// TIA Portal V15.1 export
// export: Created 2024-06-21T08:41:25.7008417Z, ExportSetting WithDefaults, DisplayName Totally Integrated Automation Portal, DisplayVersion V15.1 Update 5, DisplayName TIA Portal Openness, DisplayVersion V15.1 Update 5, DisplayName SINAMICS Startdrive Advanced, DisplayVersion V15.1, DisplayName G130, G150, S120, S150, SINAMICS MV, S210, DisplayVersion V15.1, DisplayName G110M, G120, G120C, G120D, G120P, DisplayVersion V15.1, DisplayName STEP 7 Professional, DisplayVersion V15.1 Update 5, DisplayName STEP 7 Safety, DisplayVersion V15.1, DisplayName WinCC Professional, DisplayVersion V15.1 Update 5, DisplayName SIMATIC Visualization Architect, DisplayVersion V15.1
FUNCTION "DPComPLC212" : Void   // FC261, FBD
TITLE = DPComPLC212
{ S7_Optimized_Access := 'FALSE' }
AUTHOR : VCG
FAMILY : LocFncGn
NAME : 211Intf
VERSION : 0.1
// stored: AutoNumber false, IsIECCheckEnabled false, SetENOAutomatically False, UDAEnableTagReadback false
   VAR_OUTPUT
      O_AlarmA : Bool;   // Alarm A
      O_AlarmB : Bool;   // Alarm B
      O_AlarmC : Bool;   // Alarm C
      O_AlarmD : Bool;   // Alarm D
      O_AlarmABCondition : Bool;   // Alarms resetable
      H_IAnim : Word;   // For animation of icon
   END_VAR
   VAR_TEMP
      TempInt : Int;
   END_VAR
BEGIN

REGION Network 1: **** --------------------- R228.01 --> 210CR23 --------------------- ****
END_REGION

REGION Network 2: **** 1 - Inputs **** 212A - Access Stop Request
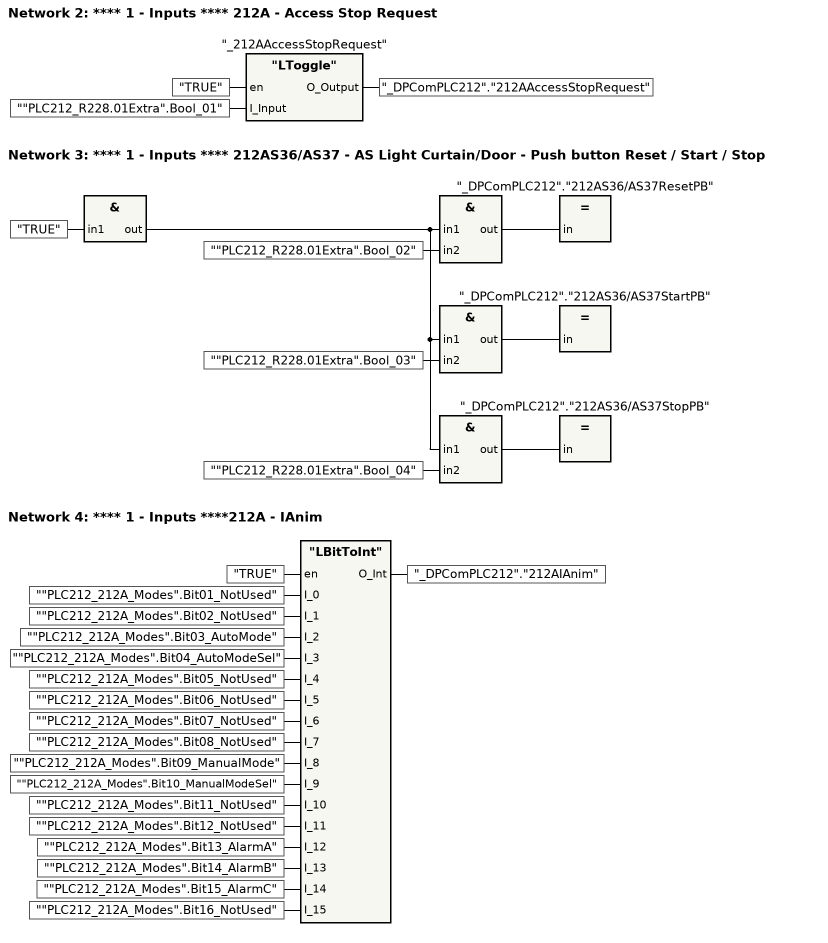
   // no checked SCL form for this network; see the picture
END_REGION

REGION Network 3: **** 1 - Inputs **** 212AS36/AS37 - AS Light Curtain/Door - Push button Reset / Start / Stop
   // no checked SCL form for this network; see the picture
END_REGION

REGION Network 4: **** 1 - Inputs ****212A - IAnim
   // no checked SCL form for this network; see the picture
END_REGION

REGION Network 5: **** 1 - Inputs **** 212A - Modes
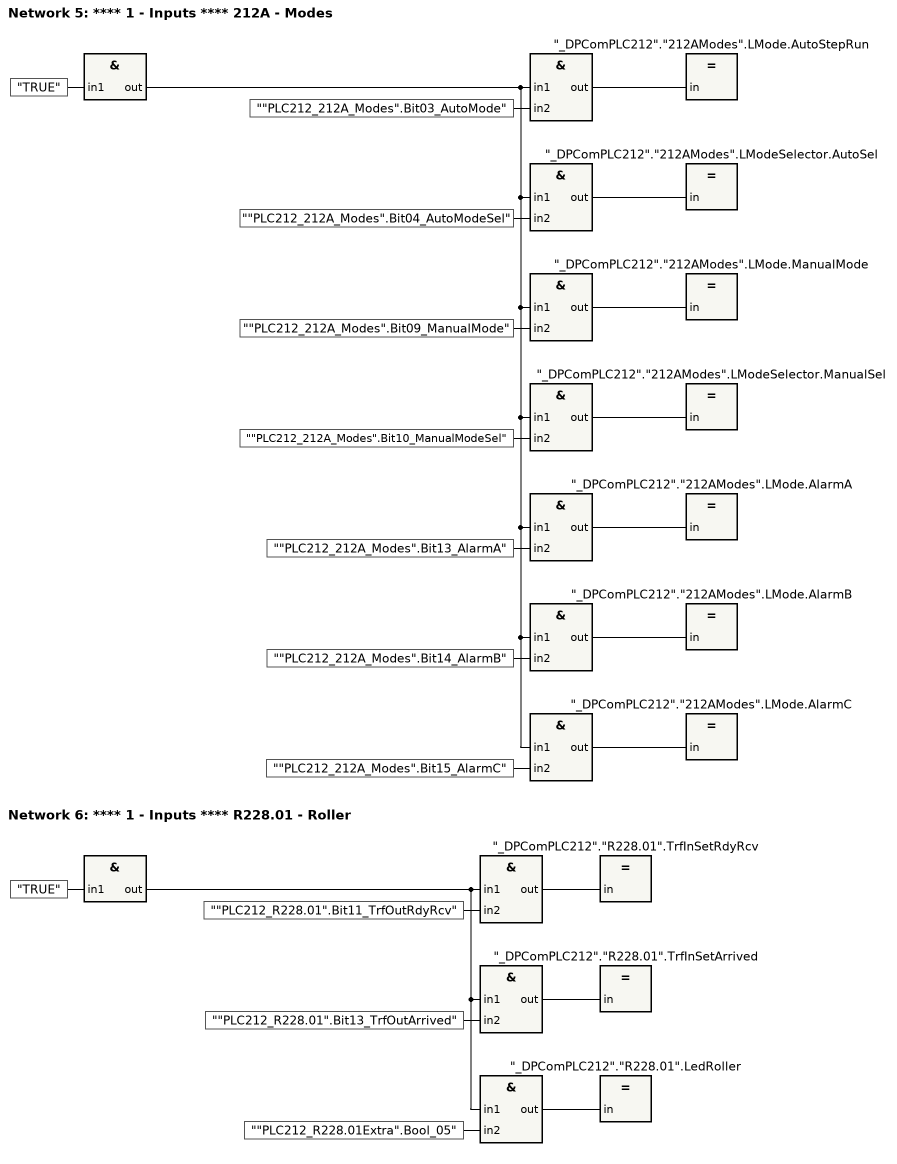
   // no checked SCL form for this network; see the picture
END_REGION

REGION Network 6: **** 1 - Inputs **** R228.01 - Roller
   // no checked SCL form for this network; see the picture
END_REGION

REGION Network 7: **** --------------------- R228.02 --> 220CR23 --------------------- ****
END_REGION

REGION Network 8: **** 1 - Inputs **** 212AS38/AS39 - AS Light Curtain/Door - Push button Reset / Start / Stop
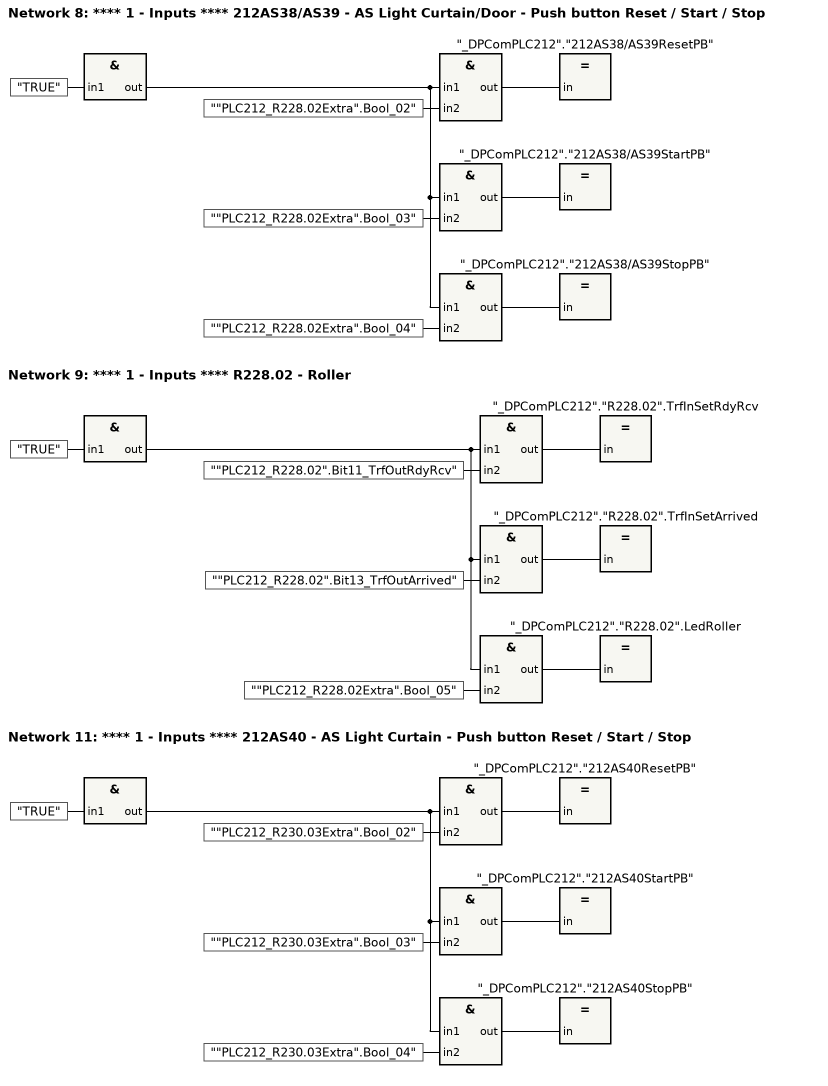
   // no checked SCL form for this network; see the picture
END_REGION

REGION Network 9: **** 1 - Inputs **** R228.02 - Roller
   // no checked SCL form for this network; see the picture
END_REGION

REGION Network 10: **** --------------------- R230.03 --> 230CA21 --------------------- ****
END_REGION

REGION Network 11: **** 1 - Inputs **** 212AS40 - AS Light Curtain - Push button Reset / Start / Stop
   // no checked SCL form for this network; see the picture
END_REGION

REGION Network 12: **** 1 - Inputs ****212D - IAnim
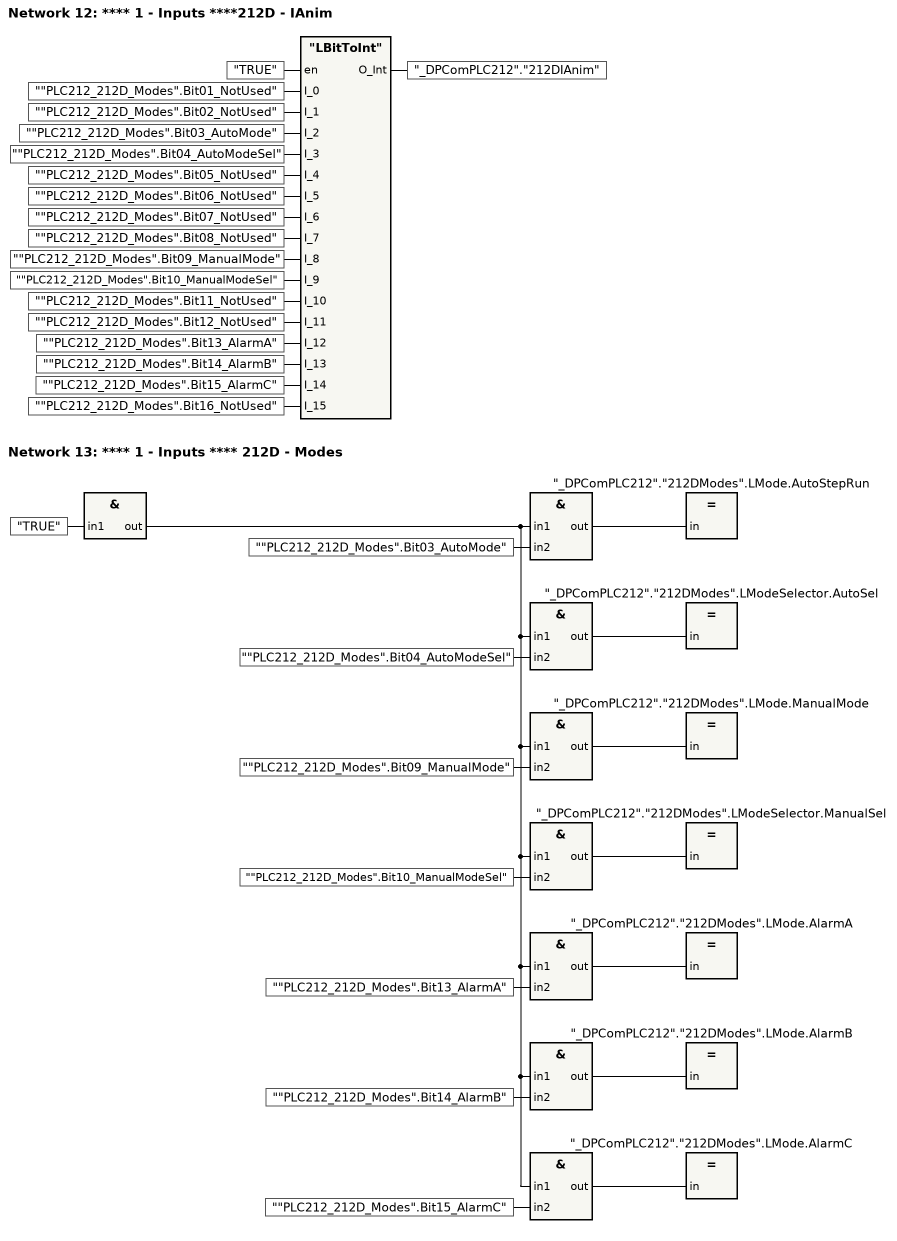
   // no checked SCL form for this network; see the picture
END_REGION

REGION Network 13: **** 1 - Inputs **** 212D - Modes
   // no checked SCL form for this network; see the picture
END_REGION

REGION Network 14: **** 1 - Inputs **** R230.03 - Roller
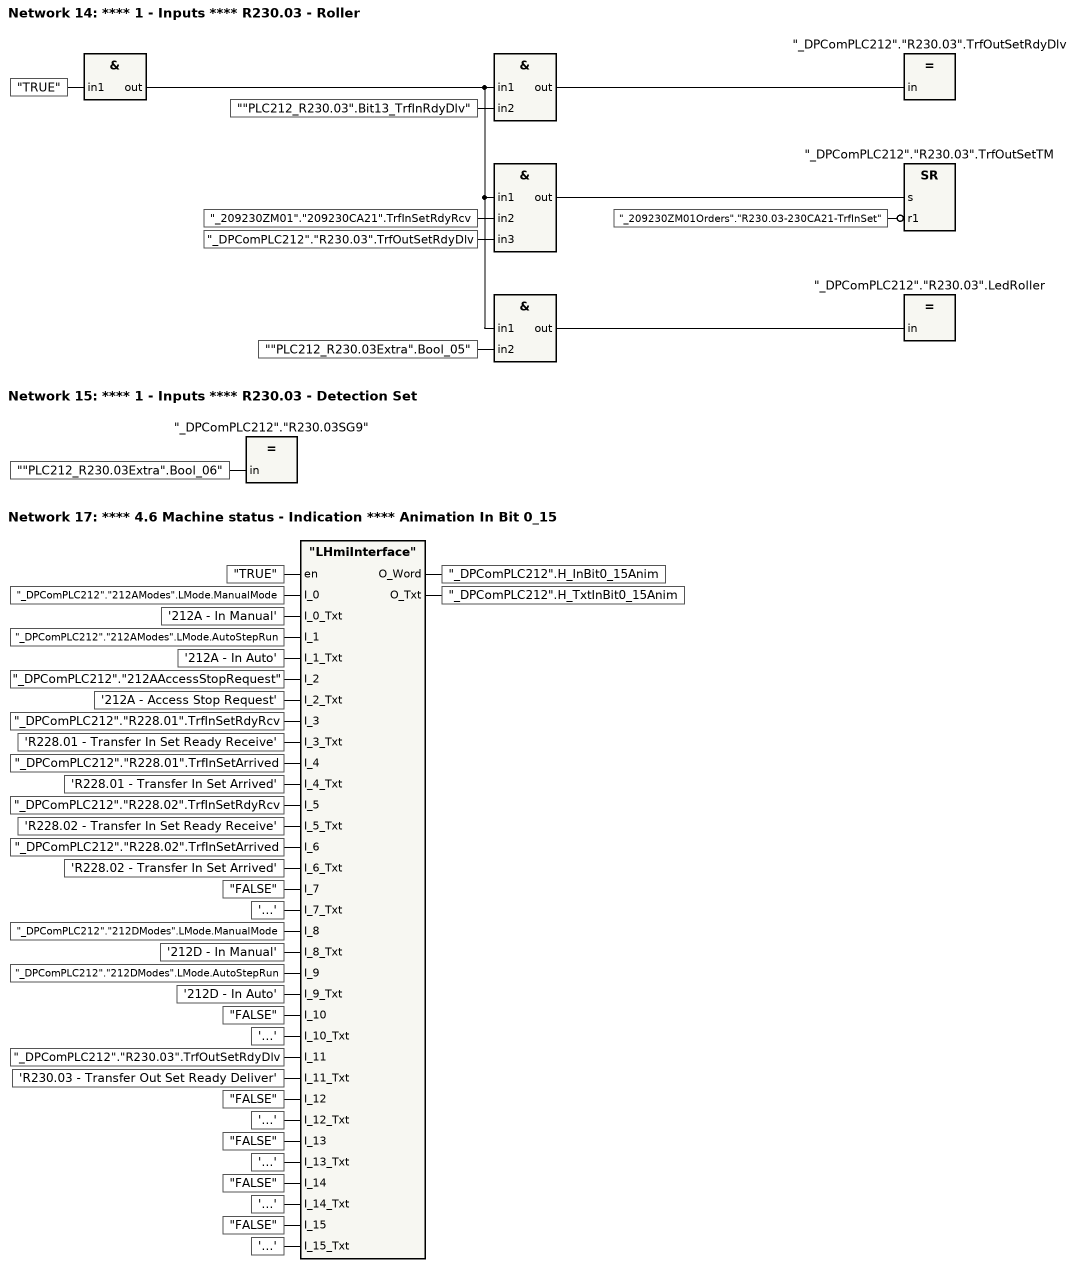
   // no checked SCL form for this network; see the picture
END_REGION

REGION Network 15: **** 1 - Inputs **** R230.03 - Detection Set
   // no checked SCL form for this network; see the picture
END_REGION

REGION Network 16: **** -------------------------------------------------- ****
END_REGION

REGION Network 17: **** 4.6 Machine status - Indication **** Animation In Bit 0_15
   // H_In0_15Anim
   IF "TRUE" THEN
       "LHmiInterface"(I_0 := "_DPComPLC212"."212AModes".LMode.ManualMode,
                       I_0_Txt := '212A - In Manual',
                       I_1 := "_DPComPLC212"."212AModes".LMode.AutoStepRun,
                       I_1_Txt := '212A - In Auto',
                       I_2 := "_DPComPLC212"."212AAccessStopRequest",
                       I_2_Txt := '212A - Access Stop Request',
                       I_3 := "_DPComPLC212"."R228.01".TrfInSetRdyRcv,
                       I_3_Txt := 'R228.01 - Transfer In Set Ready Receive',
                       I_4 := "_DPComPLC212"."R228.01".TrfInSetArrived,
                       I_4_Txt := 'R228.01 - Transfer In Set Arrived',
                       I_5 := "_DPComPLC212"."R228.02".TrfInSetRdyRcv,
                       I_5_Txt := 'R228.02 - Transfer In Set Ready Receive',
                       I_6 := "_DPComPLC212"."R228.02".TrfInSetArrived,
                       I_6_Txt := 'R228.02 - Transfer In Set Arrived',
                       I_7 := "FALSE",
                       I_7_Txt := '...',
                       I_8 := "_DPComPLC212"."212DModes".LMode.ManualMode,
                       I_8_Txt := '212D - In Manual',
                       I_9 := "_DPComPLC212"."212DModes".LMode.AutoStepRun,
                       I_9_Txt := '212D - In Auto',
                       I_10 := "FALSE",
                       I_10_Txt := '...',
                       I_11 := "_DPComPLC212"."R230.03".TrfOutSetRdyDlv,
                       I_11_Txt := 'R230.03 - Transfer Out Set Ready Deliver',
                       I_12 := "FALSE",
                       I_12_Txt := '...',
                       I_13 := "FALSE",
                       I_13_Txt := '...',
                       I_14 := "FALSE",
                       I_14_Txt := '...',
                       I_15 := "FALSE",
                       I_15_Txt := '...',
                       O_Word => "_DPComPLC212".H_InBit0_15Anim,
                       O_Txt => "_DPComPLC212".H_TxtInBit0_15Anim);
   END_IF;
END_REGION

REGION Network 18: **** 4.6 Machine status - Indication **** Animation In Bit 16_31
   // H_In16_31Anim
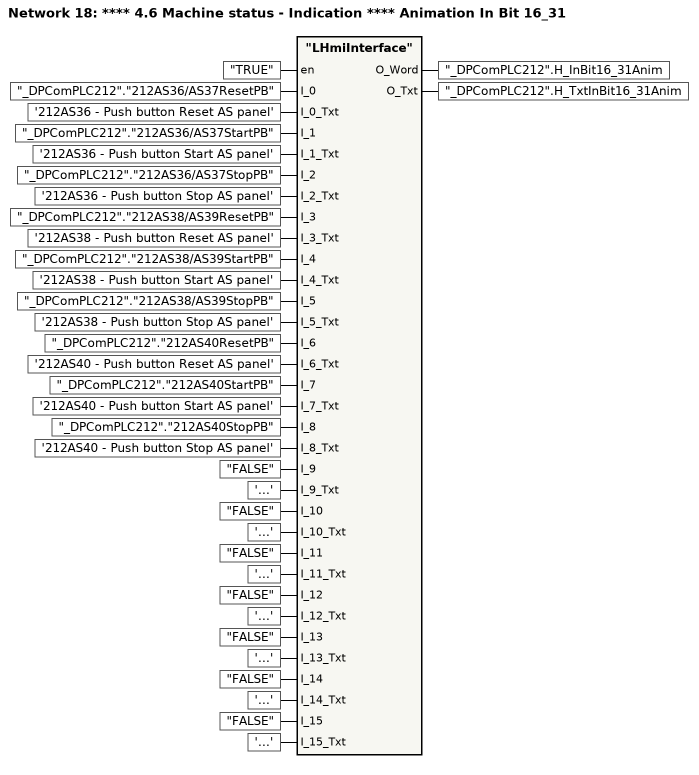
   IF "TRUE" THEN
       "LHmiInterface"(I_0 := "_DPComPLC212"."212AS36/AS37ResetPB",
                       I_0_Txt := '212AS36 - Push button Reset AS panel',
                       I_1 := "_DPComPLC212"."212AS36/AS37StartPB",
                       I_1_Txt := '212AS36 - Push button Start AS panel',
                       I_2 := "_DPComPLC212"."212AS36/AS37StopPB",
                       I_2_Txt := '212AS36 - Push button Stop AS panel',
                       I_3 := "_DPComPLC212"."212AS38/AS39ResetPB",
                       I_3_Txt := '212AS38 - Push button Reset AS panel',
                       I_4 := "_DPComPLC212"."212AS38/AS39StartPB",
                       I_4_Txt := '212AS38 - Push button Start AS panel',
                       I_5 := "_DPComPLC212"."212AS38/AS39StopPB",
                       I_5_Txt := '212AS38 - Push button Stop AS panel',
                       I_6 := "_DPComPLC212"."212AS40ResetPB",
                       I_6_Txt := '212AS40 - Push button Reset AS panel',
                       I_7 := "_DPComPLC212"."212AS40StartPB",
                       I_7_Txt := '212AS40 - Push button Start AS panel',
                       I_8 := "_DPComPLC212"."212AS40StopPB",
                       I_8_Txt := '212AS40 - Push button Stop AS panel',
                       I_9 := "FALSE",
                       I_9_Txt := '...',
                       I_10 := "FALSE",
                       I_10_Txt := '...',
                       I_11 := "FALSE",
                       I_11_Txt := '...',
                       I_12 := "FALSE",
                       I_12_Txt := '...',
                       I_13 := "FALSE",
                       I_13_Txt := '...',
                       I_14 := "FALSE",
                       I_14_Txt := '...',
                       I_15 := "FALSE",
                       I_15_Txt := '...',
                       O_Word => "_DPComPLC212".H_InBit16_31Anim,
                       O_Txt => "_DPComPLC212".H_TxtInBit16_31Anim);
   END_IF;
END_REGION

REGION Network 19: **** 4.6 Machine status - Indication **** Animation Out Bit 0_15
   // H_Out0_15Anim
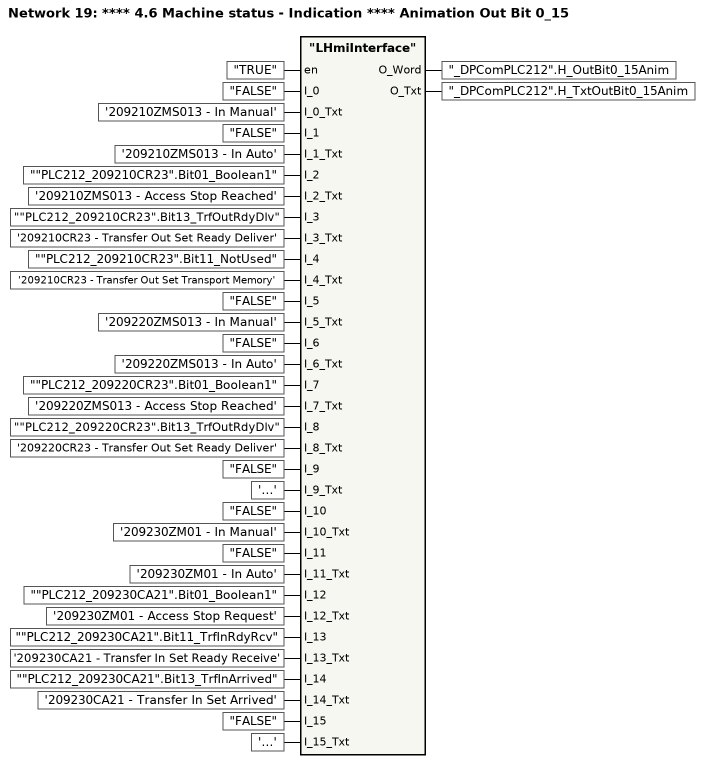
   // no checked SCL form for this network; see the picture
END_REGION

REGION Network 20: **** 4.6 Machine status - Indication **** Animation Out Bit 16_31
   // H_Out16_31Anim
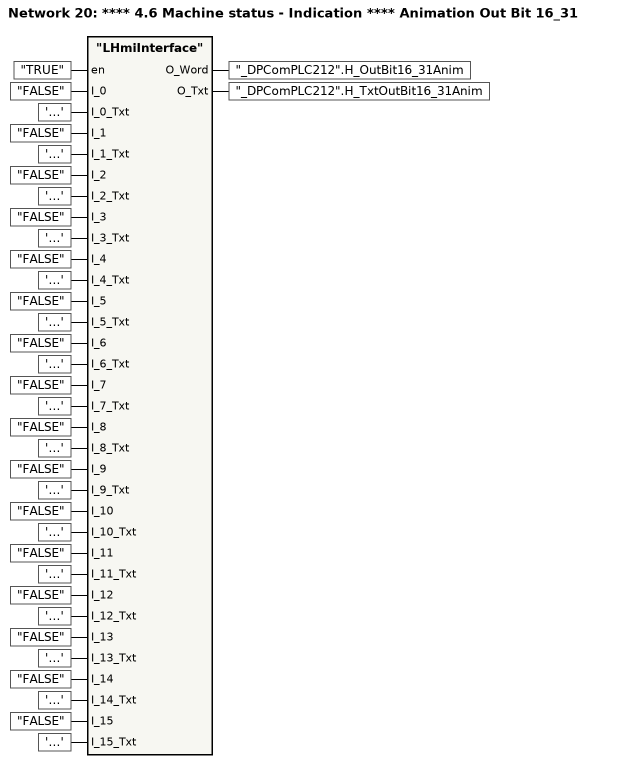
   IF "TRUE" THEN
       "LHmiInterface"(I_0 := "FALSE",
                       I_0_Txt := '...',
                       I_1 := "FALSE",
                       I_1_Txt := '...',
                       I_2 := "FALSE",
                       I_2_Txt := '...',
                       I_3 := "FALSE",
                       I_3_Txt := '...',
                       I_4 := "FALSE",
                       I_4_Txt := '...',
                       I_5 := "FALSE",
                       I_5_Txt := '...',
                       I_6 := "FALSE",
                       I_6_Txt := '...',
                       I_7 := "FALSE",
                       I_7_Txt := '...',
                       I_8 := "FALSE",
                       I_8_Txt := '...',
                       I_9 := "FALSE",
                       I_9_Txt := '...',
                       I_10 := "FALSE",
                       I_10_Txt := '...',
                       I_11 := "FALSE",
                       I_11_Txt := '...',
                       I_12 := "FALSE",
                       I_12_Txt := '...',
                       I_13 := "FALSE",
                       I_13_Txt := '...',
                       I_14 := "FALSE",
                       I_14_Txt := '...',
                       I_15 := "FALSE",
                       I_15_Txt := '...',
                       O_Word => "_DPComPLC212".H_OutBit16_31Anim,
                       O_Txt => "_DPComPLC212".H_TxtOutBit16_31Anim);
   END_IF;
END_REGION

REGION Network 21: **** 4.6 Machine status - Indication **** Animation Safety In Bit 0_15
   // H_FIn0_15Anim
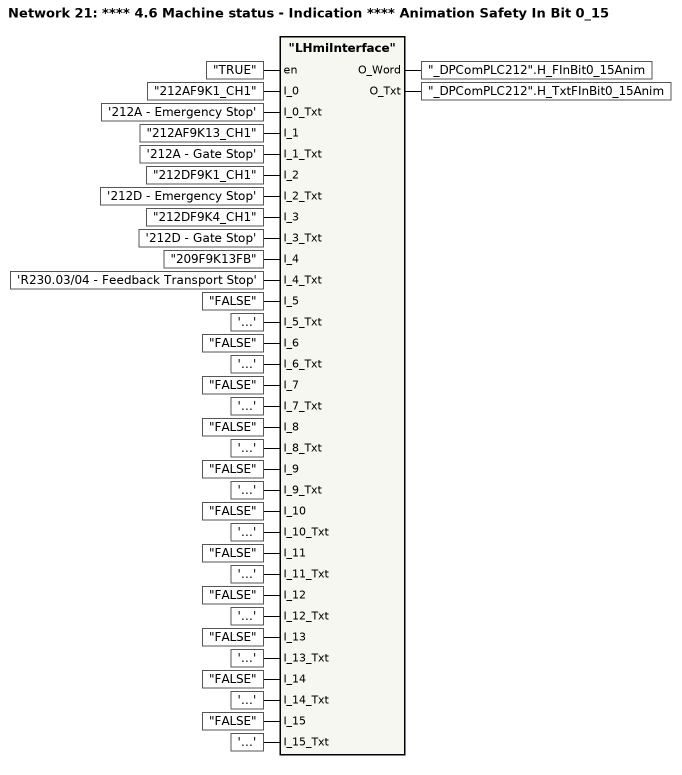
   IF "TRUE" THEN
       "LHmiInterface"(I_0 := "212AF9K1_CH1",
                       I_0_Txt := '212A - Emergency Stop',
                       I_1 := "212AF9K13_CH1",
                       I_1_Txt := '212A - Gate Stop',
                       I_2 := "212DF9K1_CH1",
                       I_2_Txt := '212D - Emergency Stop',
                       I_3 := "212DF9K4_CH1",
                       I_3_Txt := '212D - Gate Stop',
                       I_4 := "209F9K13FB",
                       I_4_Txt := 'R230.03/04 - Feedback Transport Stop',
                       I_5 := "FALSE",
                       I_5_Txt := '...',
                       I_6 := "FALSE",
                       I_6_Txt := '...',
                       I_7 := "FALSE",
                       I_7_Txt := '...',
                       I_8 := "FALSE",
                       I_8_Txt := '...',
                       I_9 := "FALSE",
                       I_9_Txt := '...',
                       I_10 := "FALSE",
                       I_10_Txt := '...',
                       I_11 := "FALSE",
                       I_11_Txt := '...',
                       I_12 := "FALSE",
                       I_12_Txt := '...',
                       I_13 := "FALSE",
                       I_13_Txt := '...',
                       I_14 := "FALSE",
                       I_14_Txt := '...',
                       I_15 := "FALSE",
                       I_15_Txt := '...',
                       O_Word => "_DPComPLC212".H_FInBit0_15Anim,
                       O_Txt => "_DPComPLC212".H_TxtFInBit0_15Anim);
   END_IF;
END_REGION

REGION Network 22: **** 4.6 Machine status - Indication **** Animation Safety Out Bit 0_15
   // H_FOut0_15Anim
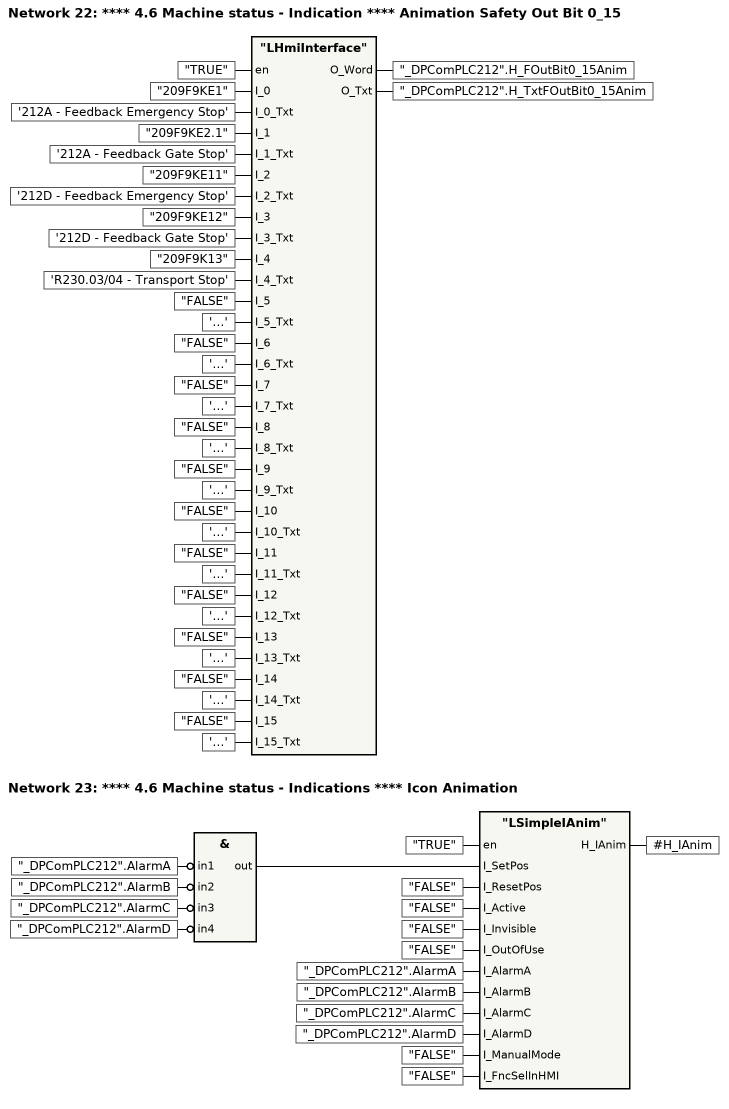
   IF "TRUE" THEN
       "LHmiInterface"(I_0 := "209F9KE1",
                       I_0_Txt := '212A - Feedback Emergency Stop',
                       I_1 := "209F9KE2.1",
                       I_1_Txt := '212A - Feedback Gate Stop',
                       I_2 := "209F9KE11",
                       I_2_Txt := '212D - Feedback Emergency Stop',
                       I_3 := "209F9KE12",
                       I_3_Txt := '212D - Feedback Gate Stop',
                       I_4 := "209F9K13",
                       I_4_Txt := 'R230.03/04 - Transport Stop',
                       I_5 := "FALSE",
                       I_5_Txt := '...',
                       I_6 := "FALSE",
                       I_6_Txt := '...',
                       I_7 := "FALSE",
                       I_7_Txt := '...',
                       I_8 := "FALSE",
                       I_8_Txt := '...',
                       I_9 := "FALSE",
                       I_9_Txt := '...',
                       I_10 := "FALSE",
                       I_10_Txt := '...',
                       I_11 := "FALSE",
                       I_11_Txt := '...',
                       I_12 := "FALSE",
                       I_12_Txt := '...',
                       I_13 := "FALSE",
                       I_13_Txt := '...',
                       I_14 := "FALSE",
                       I_14_Txt := '...',
                       I_15 := "FALSE",
                       I_15_Txt := '...',
                       O_Word => "_DPComPLC212".H_FOutBit0_15Anim,
                       O_Txt => "_DPComPLC212".H_TxtFOutBit0_15Anim);
   END_IF;
END_REGION

REGION Network 23: **** 4.6 Machine status - Indications **** Icon Animation
   // Animation for icon
   IF "TRUE" THEN
       "LSimpleIAnim"(I_SetPos := NOT "_DPComPLC212".AlarmA AND NOT "_DPComPLC212".AlarmB AND NOT "_DPComPLC212".AlarmC AND NOT "_DPComPLC212".AlarmD,
                      I_ResetPos := "FALSE",
                      I_Active := "FALSE",
                      I_Invisible := "FALSE",
                      I_OutOfUse := "FALSE",
                      I_AlarmA := "_DPComPLC212".AlarmA,
                      I_AlarmB := "_DPComPLC212".AlarmB,
                      I_AlarmC := "_DPComPLC212".AlarmC,
                      I_AlarmD := "_DPComPLC212".AlarmD,
                      I_ManualMode := "FALSE",
                      I_FncSelInHMI := "FALSE",
                      H_IAnim => #H_IAnim);
   END_IF;
END_REGION

REGION Network 24: **** 4.6 - Machine status - Indications **** Animation
   // Animation
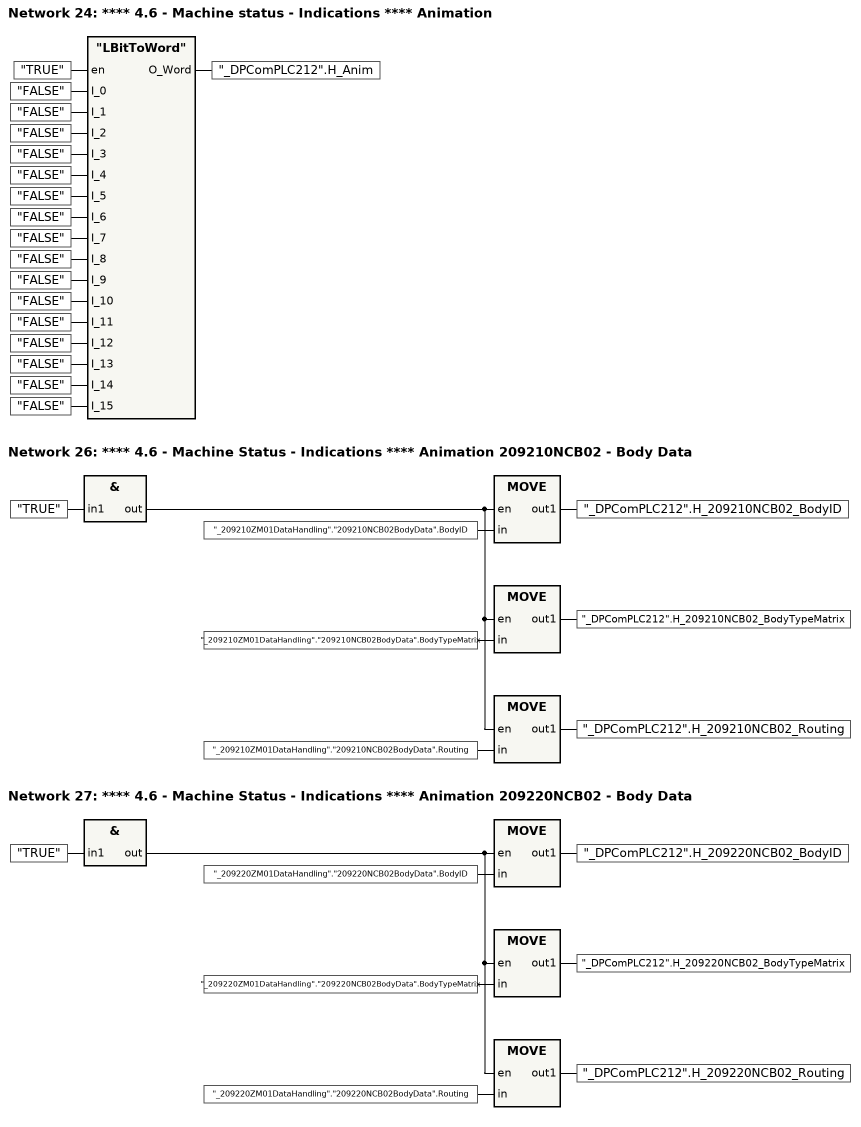
   IF "TRUE" THEN
       "LBitToWord"(I_0 := "FALSE",
                    I_1 := "FALSE",
                    I_2 := "FALSE",
                    I_3 := "FALSE",
                    I_4 := "FALSE",
                    I_5 := "FALSE",
                    I_6 := "FALSE",
                    I_7 := "FALSE",
                    I_8 := "FALSE",
                    I_9 := "FALSE",
                    I_10 := "FALSE",
                    I_11 := "FALSE",
                    I_12 := "FALSE",
                    I_13 := "FALSE",
                    I_14 := "FALSE",
                    I_15 := "FALSE",
                    O_Word => "_DPComPLC212".H_Anim);
   END_IF;
END_REGION

NETWORK
TITLE = **** 4.6 - Machine Status - Indications **** Animation DB number
// DB number
      OPN   "_DPComPLC212";
      L     DBNO;
      T     "_DPComPLC212".H_DBnr;

REGION Network 26: **** 4.6 - Machine Status - Indications **** Animation 209210NCB02 - Body Data
   IF "TRUE" THEN
       "_DPComPLC212".H_209210NCB02_BodyID := "_209210ZM01DataHandling"."209210NCB02BodyData".BodyID;
       "_DPComPLC212".H_209210NCB02_BodyTypeMatrix := "_209210ZM01DataHandling"."209210NCB02BodyData".BodyTypeMatrix;
       "_DPComPLC212".H_209210NCB02_Routing := "_209210ZM01DataHandling"."209210NCB02BodyData".Routing;
   END_IF;
END_REGION

REGION Network 27: **** 4.6 - Machine Status - Indications **** Animation 209220NCB02 - Body Data
   IF "TRUE" THEN
       "_DPComPLC212".H_209220NCB02_BodyID := "_209220ZM01DataHandling"."209220NCB02BodyData".BodyID;
       "_DPComPLC212".H_209220NCB02_BodyTypeMatrix := "_209220ZM01DataHandling"."209220NCB02BodyData".BodyTypeMatrix;
       "_DPComPLC212".H_209220NCB02_Routing := "_209220ZM01DataHandling"."209220NCB02BodyData".Routing;
   END_IF;
END_REGION

REGION Network 28: **** 7.1 - Submodules - NonMachine **** Check DP/DP Coupler (Live Bit)
   // Check DP/DP Coupler (Live Bit)
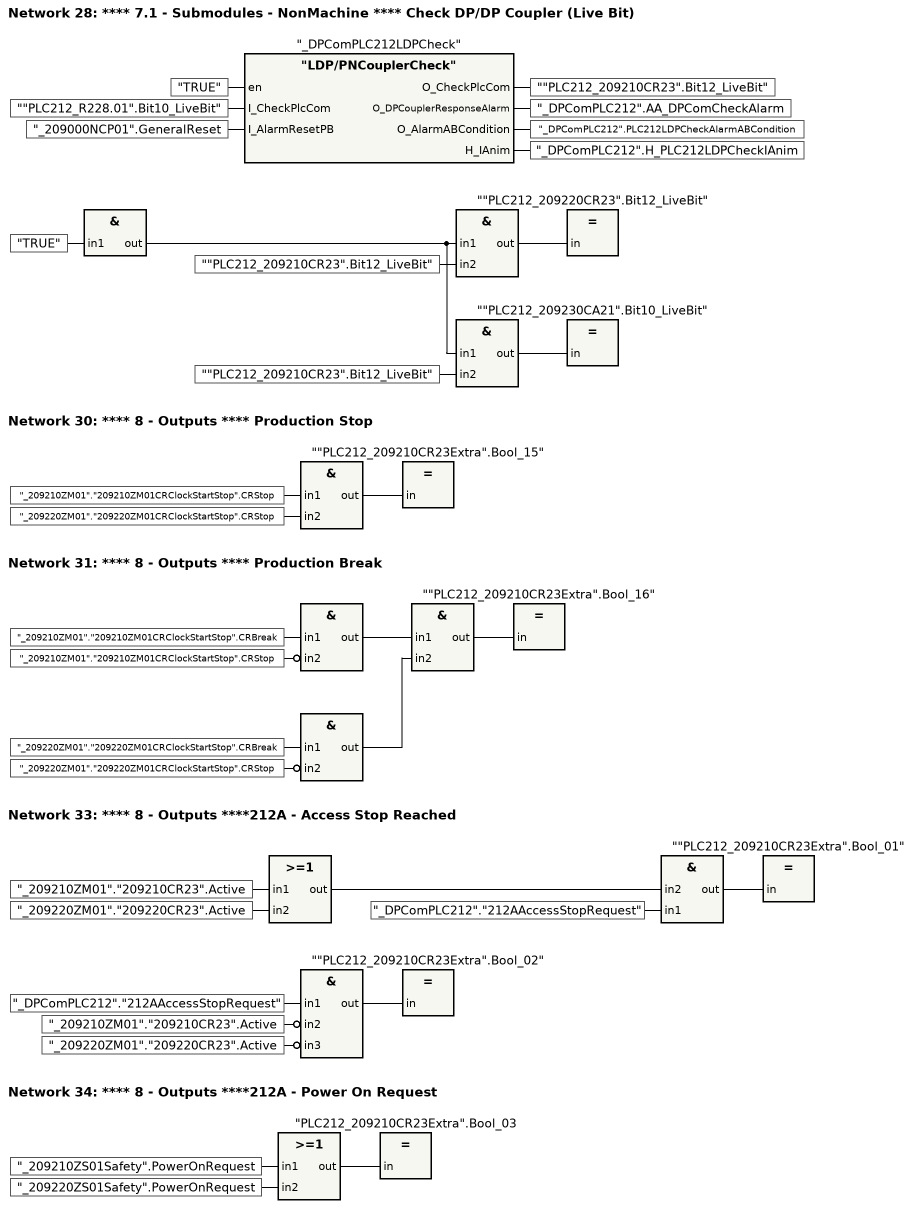
   // no checked SCL form for this network; see the picture
END_REGION

REGION Network 29: **** --------------------- Global --------------------- ****
END_REGION

REGION Network 30: **** 8 - Outputs **** Production Stop
   // no checked SCL form for this network; see the picture
END_REGION

REGION Network 31: **** 8 - Outputs **** Production Break
   // no checked SCL form for this network; see the picture
END_REGION

REGION Network 32: **** --------------------- 210CR23 --> R228.01 --------------------- ****
END_REGION

REGION Network 33: **** 8 - Outputs ****212A - Access Stop Reached
   // no checked SCL form for this network; see the picture
END_REGION

REGION Network 34: **** 8 - Outputs ****212A - Power On Request
   "PLC212_209210CR23Extra".Bool_03 := "_209210ZS01Safety".PowerOnRequest OR "_209220ZS01Safety".PowerOnRequest;
END_REGION

REGION Network 35: **** 8 - Outputs **** 209210ZMS013 - Modes
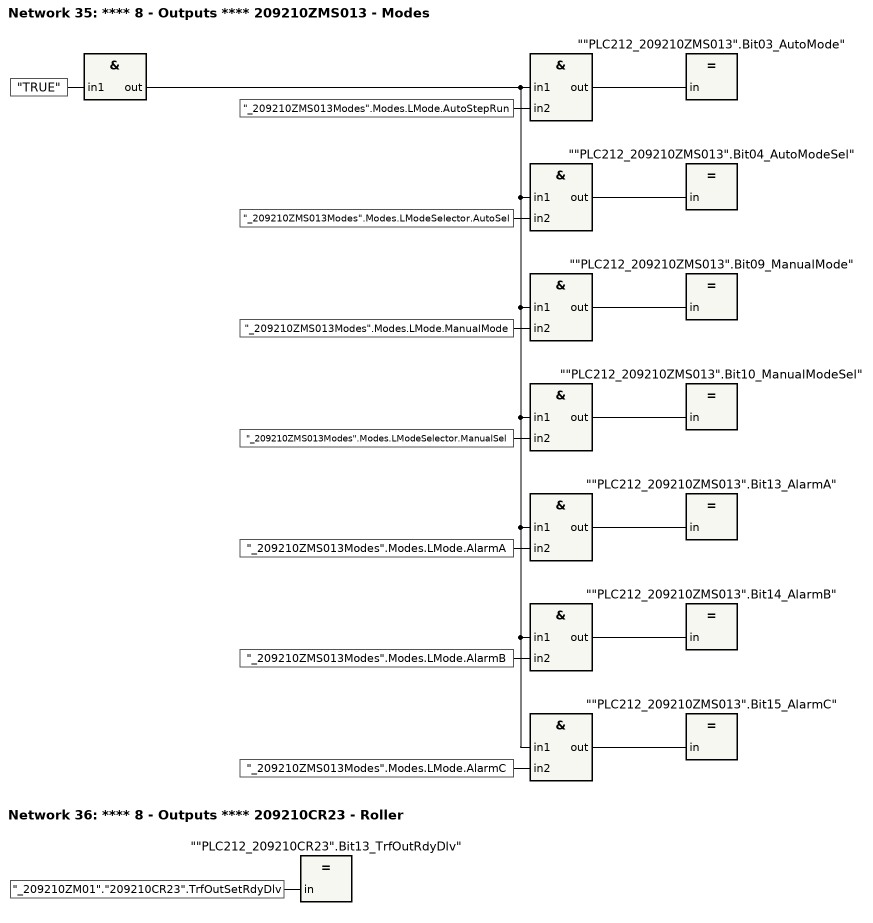
   // no checked SCL form for this network; see the picture
END_REGION

REGION Network 36: **** 8 - Outputs **** 209210CR23 - Roller
   // no checked SCL form for this network; see the picture
END_REGION

REGION Network 37: **** 8 - Outputs **** 209210NCB02 - Body Data
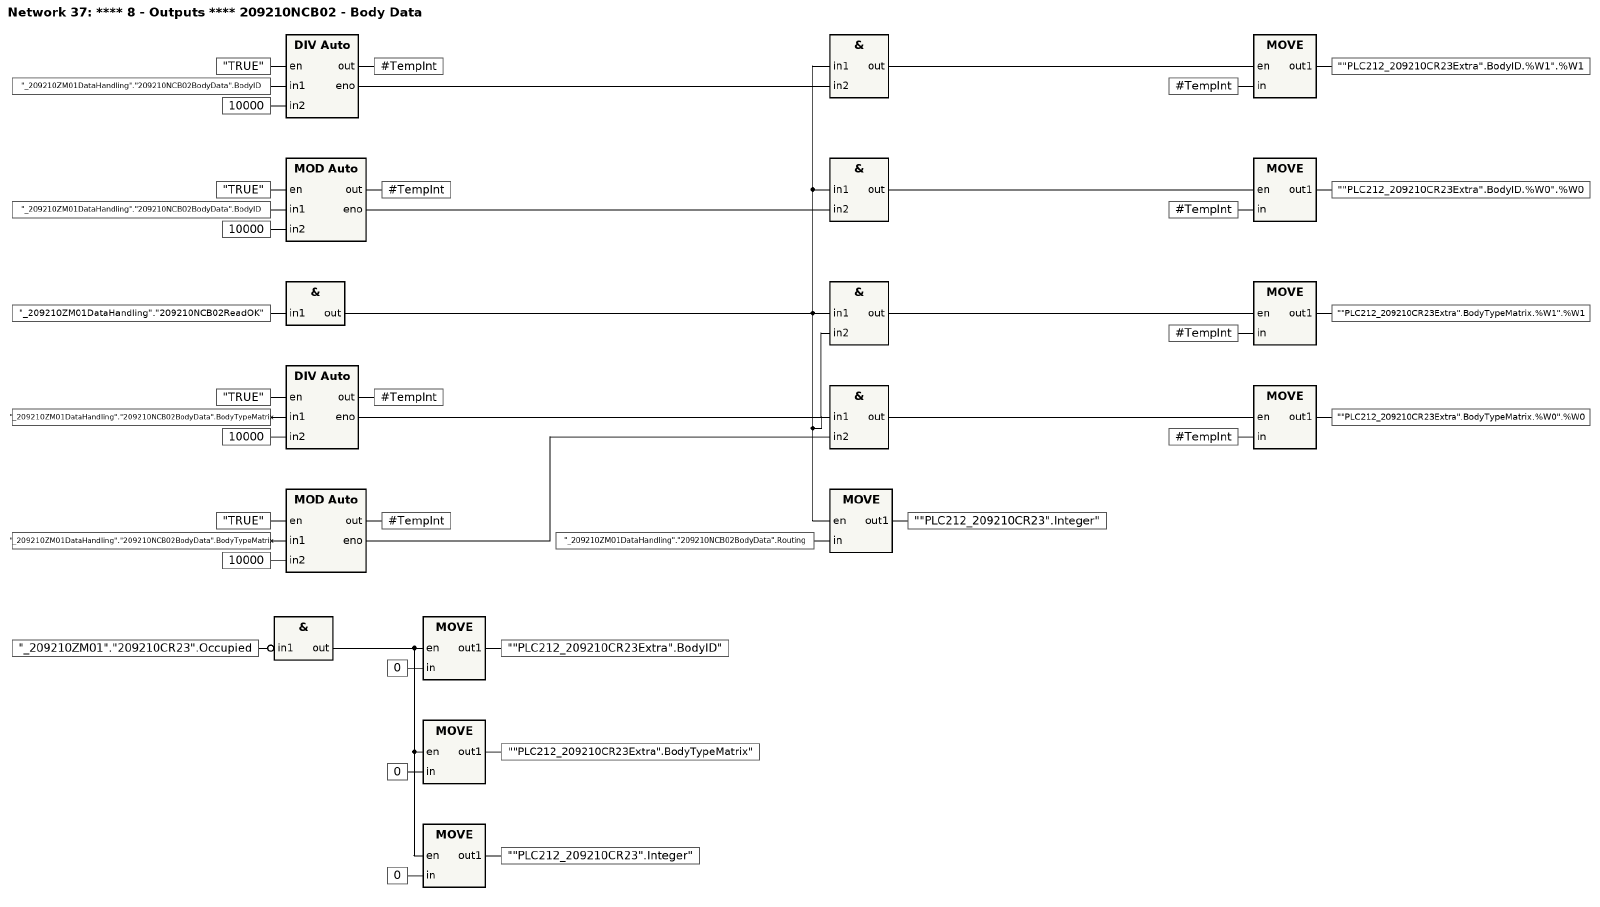
   // no checked SCL form for this network; see the picture
END_REGION

REGION Network 38: **** --------------------- 220CR23 --> R228.02 --------------------- ****
END_REGION

REGION Network 39: **** 8 - Outputs **** 209220ZMS013 - Modes
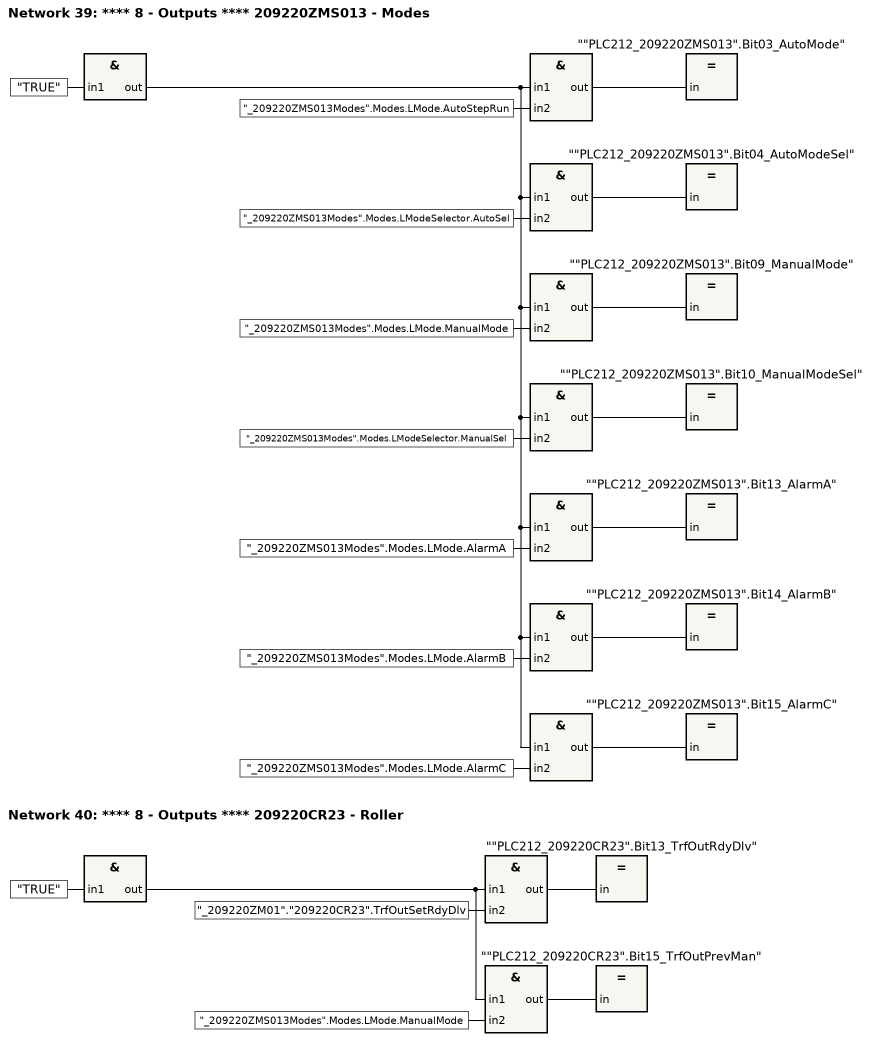
   // no checked SCL form for this network; see the picture
END_REGION

REGION Network 40: **** 8 - Outputs **** 209220CR23 - Roller
   // no checked SCL form for this network; see the picture
END_REGION

REGION Network 41: **** 8 - Outputs **** 209220NCB02 - Body Data
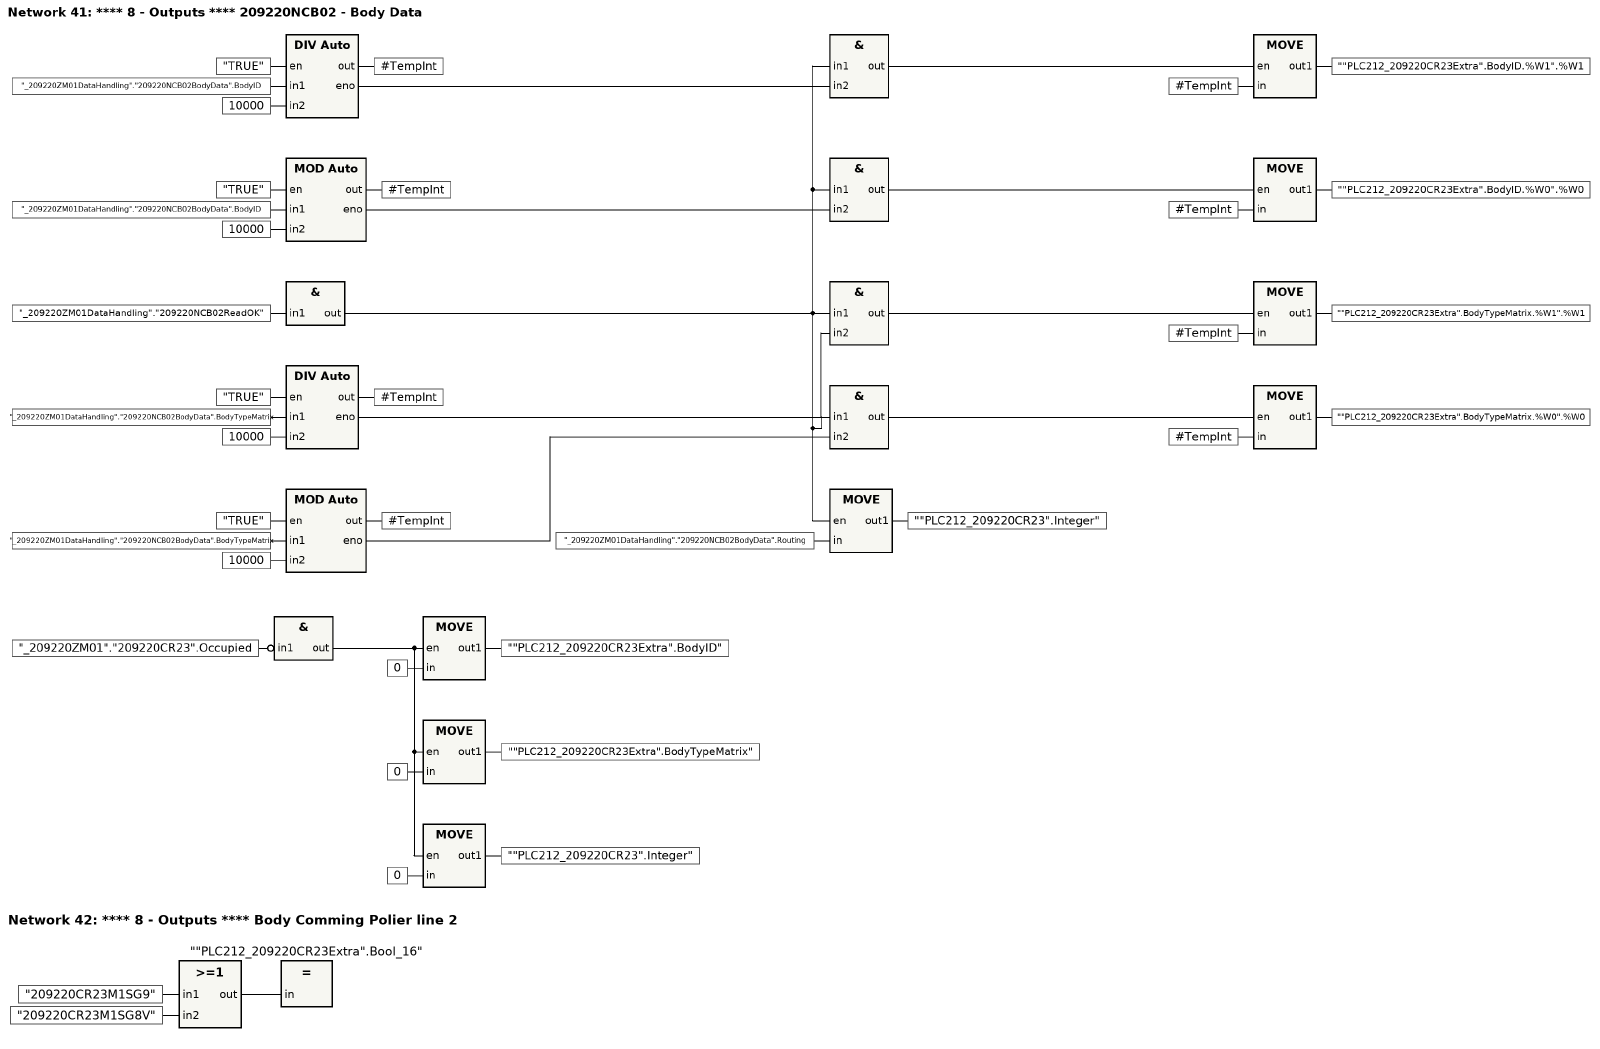
   // no checked SCL form for this network; see the picture
END_REGION

REGION Network 42: **** 8 - Outputs **** Body Comming Polier line 2
   // no checked SCL form for this network; see the picture
END_REGION

REGION Network 43: **** --------------------- 230CA21 --> R230.03 --------------------- ****
END_REGION

REGION Network 44: **** 8 - Outputs **** 209230ZM01 - Modes
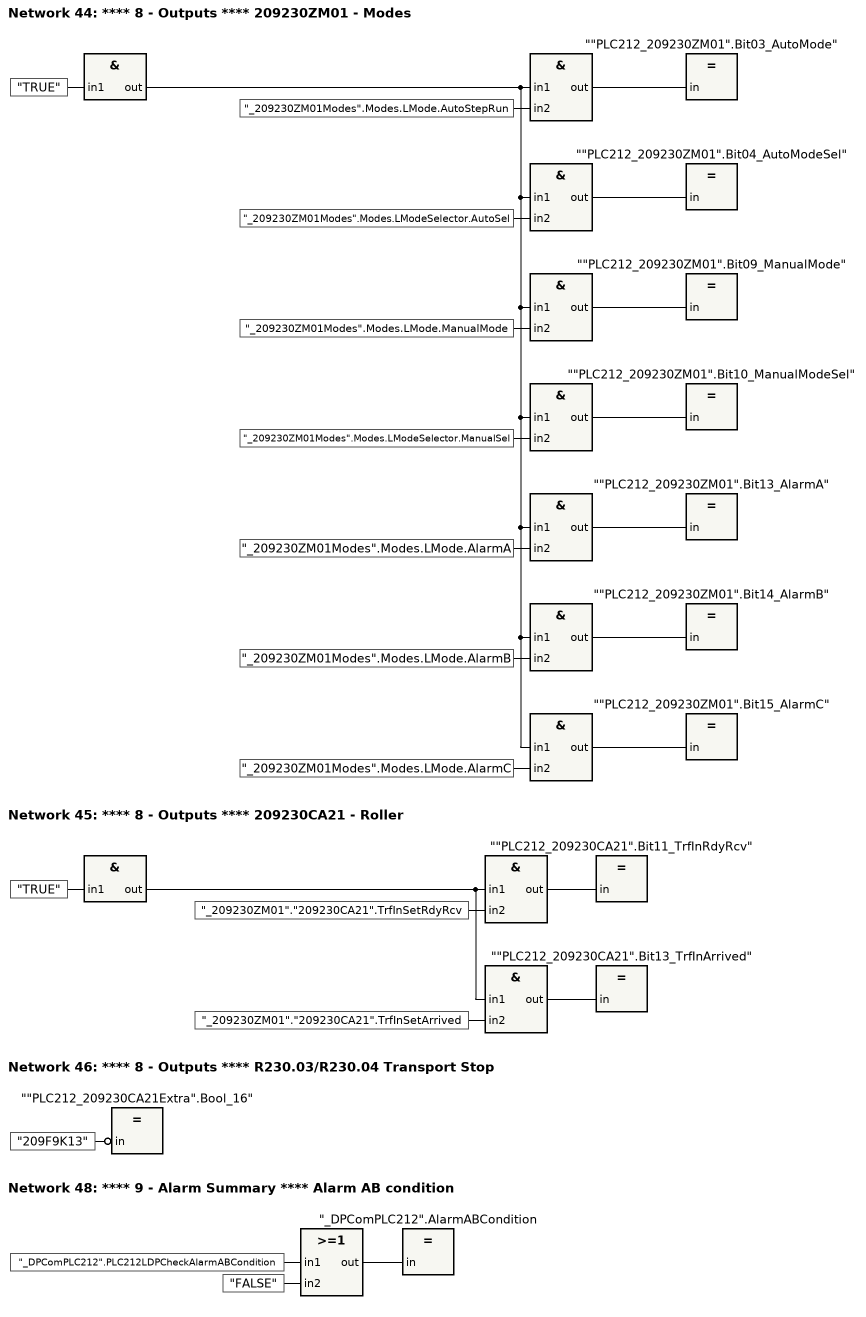
   // no checked SCL form for this network; see the picture
END_REGION

REGION Network 45: **** 8 - Outputs **** 209230CA21 - Roller
   // no checked SCL form for this network; see the picture
END_REGION

REGION Network 46: **** 8 - Outputs **** R230.03/R230.04 Transport Stop
   // no checked SCL form for this network; see the picture
END_REGION

REGION Network 47: **** -------------------------------------------------- ****
END_REGION

REGION Network 48: **** 9 - Alarm Summary **** Alarm AB condition
   // Alarm AB condition
   "_DPComPLC212".AlarmABCondition := "_DPComPLC212".PLC212LDPCheckAlarmABCondition OR "FALSE";
END_REGION

REGION Network 49: **** 9 - Alarm Summary **** Alarm A
   // Summary of alarms A
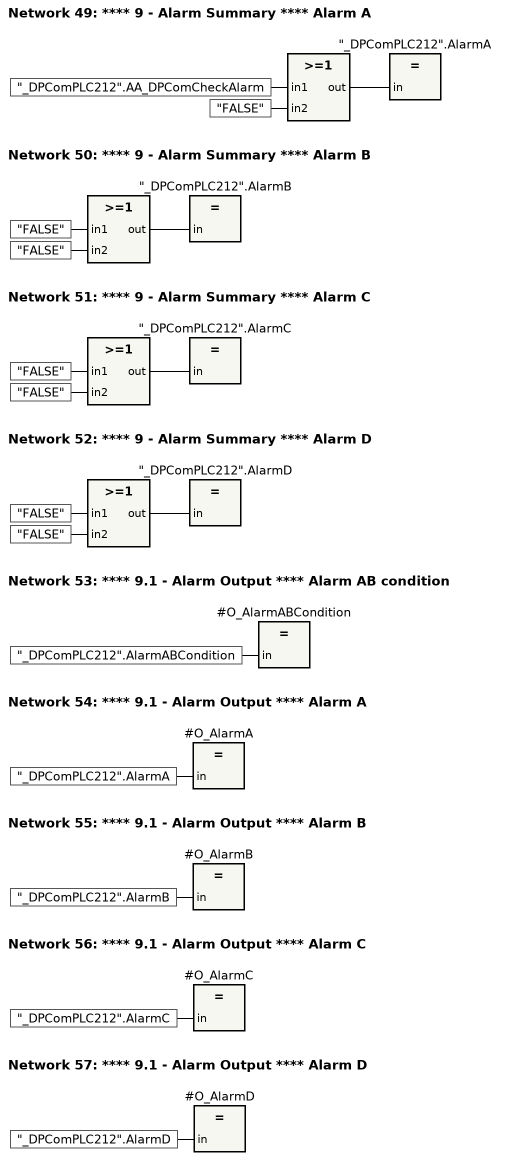
   "_DPComPLC212".AlarmA := "_DPComPLC212".AA_DPComCheckAlarm OR "FALSE";
END_REGION

REGION Network 50: **** 9 - Alarm Summary **** Alarm B
   // Summary of alarms B
   "_DPComPLC212".AlarmB := "FALSE" OR "FALSE";
END_REGION

REGION Network 51: **** 9 - Alarm Summary **** Alarm C
   // Summary of alarms C
   "_DPComPLC212".AlarmC := "FALSE" OR "FALSE";
END_REGION

REGION Network 52: **** 9 - Alarm Summary **** Alarm D
   // Summary of alarms D
   "_DPComPLC212".AlarmD := "FALSE" OR "FALSE";
END_REGION

REGION Network 53: **** 9.1 - Alarm Output **** Alarm AB condition
   // Alarm AB condition
   #O_AlarmABCondition := "_DPComPLC212".AlarmABCondition;
END_REGION

REGION Network 54: **** 9.1 - Alarm Output **** Alarm A
   // Summary of alarms A
   #O_AlarmA := "_DPComPLC212".AlarmA;
END_REGION

REGION Network 55: **** 9.1 - Alarm Output **** Alarm B
   // Summary of alarms B
   #O_AlarmB := "_DPComPLC212".AlarmB;
END_REGION

REGION Network 56: **** 9.1 - Alarm Output **** Alarm C
   // Summary of alarms C
   #O_AlarmC := "_DPComPLC212".AlarmC;
END_REGION

REGION Network 57: **** 9.1 - Alarm Output **** Alarm D
   // Summary of alarms D
   #O_AlarmD := "_DPComPLC212".AlarmD;
END_REGION

REGION Network 58: **** 9.2 - Alarm DWord**** Alarm To DWord
   // Alarm Word
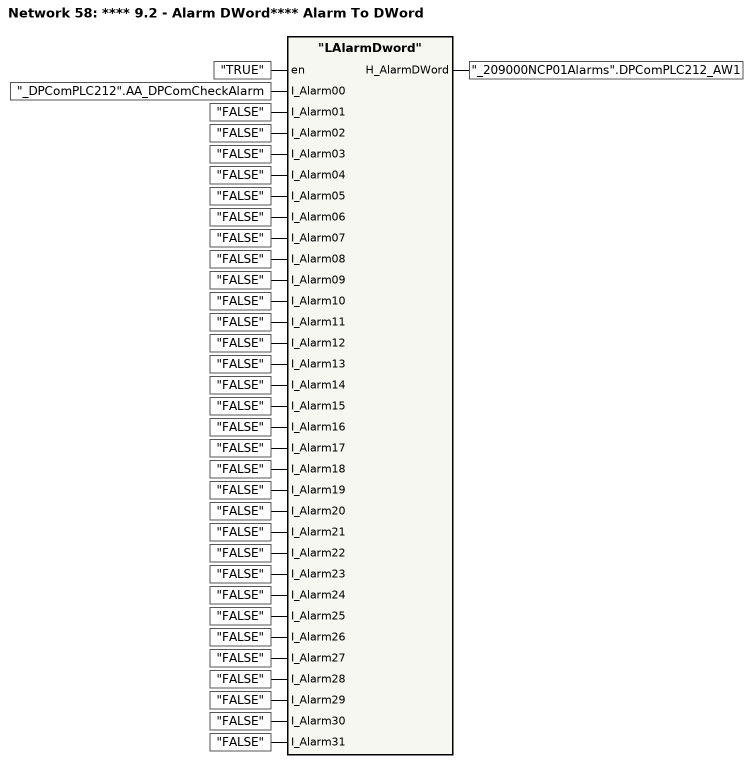
   IF "TRUE" THEN
       "LAlarmDword"(I_Alarm00 := "_DPComPLC212".AA_DPComCheckAlarm,
                     I_Alarm01 := "FALSE",
                     I_Alarm02 := "FALSE",
                     I_Alarm03 := "FALSE",
                     I_Alarm04 := "FALSE",
                     I_Alarm05 := "FALSE",
                     I_Alarm06 := "FALSE",
                     I_Alarm07 := "FALSE",
                     I_Alarm08 := "FALSE",
                     I_Alarm09 := "FALSE",
                     I_Alarm10 := "FALSE",
                     I_Alarm11 := "FALSE",
                     I_Alarm12 := "FALSE",
                     I_Alarm13 := "FALSE",
                     I_Alarm14 := "FALSE",
                     I_Alarm15 := "FALSE",
                     I_Alarm16 := "FALSE",
                     I_Alarm17 := "FALSE",
                     I_Alarm18 := "FALSE",
                     I_Alarm19 := "FALSE",
                     I_Alarm20 := "FALSE",
                     I_Alarm21 := "FALSE",
                     I_Alarm22 := "FALSE",
                     I_Alarm23 := "FALSE",
                     I_Alarm24 := "FALSE",
                     I_Alarm25 := "FALSE",
                     I_Alarm26 := "FALSE",
                     I_Alarm27 := "FALSE",
                     I_Alarm28 := "FALSE",
                     I_Alarm29 := "FALSE",
                     I_Alarm30 := "FALSE",
                     I_Alarm31 := "FALSE",
                     H_AlarmDWord => "_209000NCP01Alarms".DPComPLC212_AW1);
   END_IF;
END_REGION
END_FUNCTION
